FUNCTION_BLOCK GET_TABLE_VALUE (* Gets a value from a table *)
  (* Standard: 61499-2 *)
  (* Version 1.0, 27-05-12, GASR, Universidade do Estado de Santa Catarina *)
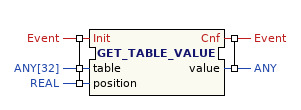
  EVENT_INPUT
    Init WITH table, position;
  END_EVENT
  EVENT_OUTPUT
    Cnf WITH value;
  END_EVENT
  VAR_INPUT
    table : ARRAY [0..31] OF ANY;
    position : REAL;
  END_VAR
  VAR_OUTPUT
    value : ANY;
  END_VAR
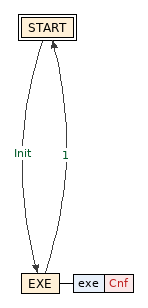
  EC_STATES
    START;
    EXE : exe -> Cnf;
  END_STATES
  EC_TRANSITIONS
    START TO EXE := Init;
    EXE TO START := 1;
  END_TRANSITIONS
  ALGORITHM exe IN Lua:
value = table[ position ]
  END_ALGORITHM
END_FUNCTION_BLOCK
